// TIA Portal V16 export
// export: Created 2025-08-01T13:37:58.9722263Z, ExportSetting WithDefaults, DisplayName Totally Integrated Automation Portal, DisplayVersion V16, DisplayName TIA Portal Version Control Interface, DisplayVersion V16, DisplayName TIA Portal Openness, DisplayVersion V16, DisplayName STEP 7 Professional, DisplayVersion V16, DisplayName STEP 7 Safety, DisplayVersion V16, DisplayName WinCC Advanced, DisplayVersion V16
FUNCTION_BLOCK "2in-1out_Block"   // FB6, FBD
VERSION : 0.1
// stored: AutoNumber true, IsIECCheckEnabled true, UDAEnableTagReadback false
   VAR_INPUT
      "Input Contact 1" : Bool;
      "Input Contact 2" : Bool;
   END_VAR
   VAR_OUTPUT
      "Output Contact 1" : Bool;
   END_VAR
BEGIN

REGION Network 1: Network Default
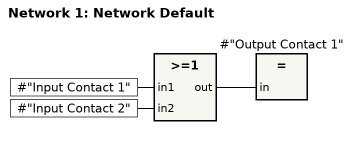
   #"Output Contact 1" := #"Input Contact 1" OR #"Input Contact 2";
END_REGION
END_FUNCTION_BLOCK
